TYPE ST_CtrlInCraneXover :
STRUCT
	ExternalDisable			: BOOL; // Disable takeover/handover externally
END_STRUCT
END_TYPE

(* stored: Version 1.1.0.1, ProductVersion 3.1.4024.9
   DUT ST_CtrlInCraneXover: Id {c64d6490-9752-4090-866e-bc499652f635} *)
